// Mitsubishi GX Works2 project: 시퀀스 예제 2_3   PLC: Q03UDV

PROGRAM MAIN
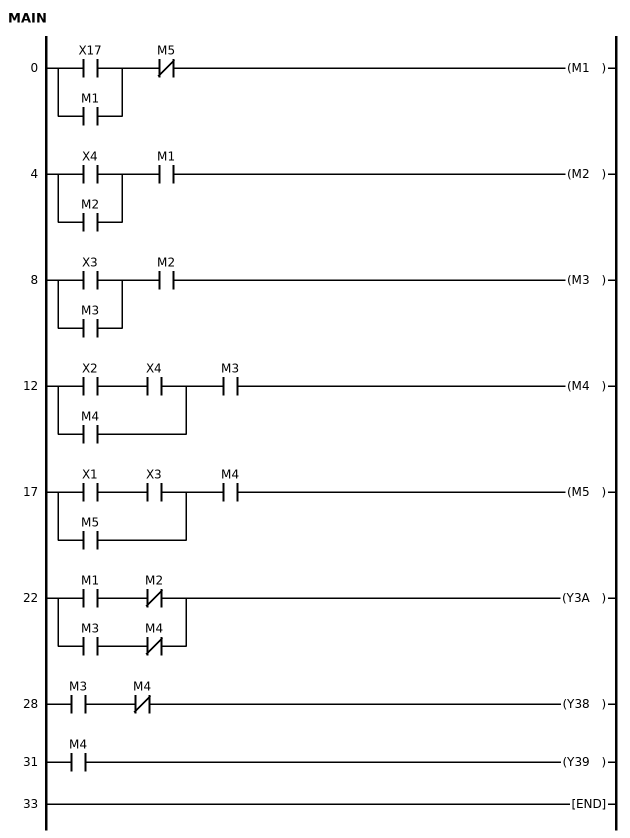
0     LD      X17
      OR      M1
      ANI     M5
      OUT     M1
4     LD      X4
      OR      M2
      AND     M1
      OUT     M2
8     LD      X3
      OR      M3
      AND     M2
      OUT     M3
12    LD      X2
      AND     X4
      OR      M4
      AND     M3
      OUT     M4
17    LD      X1
      AND     X3
      OR      M5
      AND     M4
      OUT     M5
22    LD      M1
      ANI     M2
      LD      M3
      ANI     M4
      ORB
      OUT     Y3A
28    LD      M3
      ANI     M4
      OUT     Y38
31    LD      M4
      OUT     Y39
33    END
END_PROGRAM
